{attribute addProperty BoxType "EL6001-0000-0020"}
{attribute addProperty Id "Transmit_requestBOOL81Receive_acceptedBOOL81Init_requestBOOL81Send_continuousBOOL81Output_lengthUSINT81"}
{attribute addProperty CRC "1262645546"}
{attribute addProperty SizeInBites "40"}
{attribute addProperty SizeInBytes "5"}
TYPE Ctrl_4B42712A :
STRUCT
	{attribute addProperty Name "Transmit_request"}
	Transmit_request : BOOL;
	{attribute addProperty Name "Receive_accepted"}
	Receive_accepted : BOOL;
	{attribute addProperty Name "Init_request"}
	Init_request : BOOL;
	{attribute addProperty Name "Send_continuous"}
	Send_continuous : BOOL;
	{attribute addProperty Name "Output_length"}
	Output_length : USINT;
END_STRUCT
END_TYPE

(* stored: Version 1.2.0.0, ProductVersion 3.1.4024.9
   DUT Ctrl_4B42712A: Id {7eb5c5d9-d554-4360-9953-9e724f3da656} *)
